// TwinCAT 3 PLC project Plc
// ProgramVersion: 3.1.4024.0
// libraries:
//   Tc2_Standard, * (Beckhoff Automation GmbH)
//   Tc2_System, * (Beckhoff Automation GmbH)
//   Tc3_Module, * (Beckhoff Automation GmbH)
// project tree:
//   / PlcTask.TcTTO
//   POUs/ MAIN.TcPOU, PRG_Testing.TcPOU
//   Utility/Actuator/ FB_Cylinder.TcPOU, FB_Cylinder_DoubleActing.TcPOU, FB_Cylinder_SingleActing.TcPOU
//   Utility/Sensor/ FB_Sensor_NC.TcPOU, FB_Sensor_NO.TcPOU
// real-time tasks:
//   TASK PlcTask: cycle T#10ms, priority 20, ADS port 350

CONFIGURATION Plc
    RESOURCE PLC ON TwinCAT3
        TASK PlcTask(INTERVAL := T#10ms, PRIORITY := 20);
        PROGRAM MAIN WITH PlcTask : MAIN;
    END_RESOURCE
END_CONFIGURATION

// ---- POUs/MAIN.TcPOU
PROGRAM MAIN
VAR
END_VAR

PRG_Testing();

END_PROGRAM

// ---- POUs/PRG_Testing.TcPOU
PROGRAM PRG_Testing
VAR
	fbCylinder_DoubleActing: FB_Cylinder_DoubleActing;
	fbCylinder_SingleActing: FB_Cylinder_SingleActing;
END_VAR


	fbCylinder_SingleActing(
	Start:= , 
	Extend:= , 
	Retract:= , 
	SensorExtended:= , 
	SensorRetracted:= , 
	EmergencyStop:= , 
	ExtendTime:= , 
	RetractTime:= , 
	Error=> , 
	ErrorCode=> , 
	Extend_RetractValve=> );
	
	fbCylinder_DoubleActing(
	Start:= , 
	Extend:= , 
	Retract:= , 
	SensorExtended:= , 
	SensorRetracted:= , 
	EmergencyStop:= , 
	ExtendTime:= , 
	RetractTime:= , 
	Error=> , 
	ErrorCode=> , 
	ExtendValve=> , 
	RetractValve=> );

END_PROGRAM

// ---- Utility/Actuator/FB_Cylinder_DoubleActing.TcPOU
FUNCTION_BLOCK FB_Cylinder_DoubleActing EXTENDS FB_Cylinder
VAR_INPUT
END_VAR
VAR_OUTPUT
    ExtendValve: BOOL;      // Valve output to extend the cylinder
    RetractValve: BOOL;     // Valve output to retract the cylinder	
END_VAR
VAR
END_VAR


	ExtendValve		:=	_ExtendValve;
	RetractValve	:=	_RetractValve;

END_FUNCTION_BLOCK

// ---- Utility/Actuator/FB_Cylinder.TcPOU
FUNCTION_BLOCK FB_Cylinder
VAR_INPUT
    Start: BOOL;                // Start signal
    Extend: BOOL;               // Extend signal
    Retract: BOOL;              // Retract signal
    SensorExtended: BOOL;       // Feedback from fully extended position sensor
    SensorRetracted: BOOL;      // Feedback from fully retracted position sensor
    EmergencyStop: BOOL;        // Emergency stop signal
    ExtendTime: TIME := T#5S;   // Time allowed to fully extend
    RetractTime: TIME := T#5S;  // Time allowed to fully retract
END_VAR

VAR_OUTPUT
    Error: BOOL;            // Error flag
    ErrorCode: INT;         // Error code for different fault conditions
END_VAR

VAR
    State: INT := 0;        // State variable for the state machine
    Timer: TON;             // Timer instance for timeouts
    _ExtendValve: BOOL;      // Valve output to extend the cylinder
    _RetractValve: BOOL;     // Valve output to retract the cylinder
END_VAR

	
	
	// State Machine Logic
	CASE State OF
		0: // Idle
			_ExtendValve := FALSE;
			_RetractValve := FALSE;
			Error := FALSE;
			ErrorCode := 0;
			
			IF EmergencyStop THEN
				State := 7; // Go to emergency stop state
			ELSIF Start THEN
				IF (Extend AND Retract) THEN
					Error := TRUE;
					ErrorCode := 1; // Invalid input (simultaneous Extend and Retract)
					State := 5; // Go to error state
				ELSIF Extend THEN
					IF NOT SensorExtended THEN
						State := 1; // Go to extend state if not already extended
					ELSE
						Error := TRUE;
						ErrorCode := 2; // Attempt to extend when already extended
						State := 5; // Go to error state
					END_IF
				ELSIF Retract THEN
					IF NOT SensorRetracted THEN
						State := 3; // Go to retract state if not already retracted
					ELSE
						Error := TRUE;
						ErrorCode := 3; // Attempt to retract when already retracted
						State := 5; // Go to error state
					END_IF
				END_IF
			END_IF
		
		1: // Extending
			_ExtendValve := TRUE;
			_RetractValve := FALSE;
			
			IF EmergencyStop THEN
				State := 7; // Go to emergency stop state
			ELSIF SensorExtended THEN
				State := 2; // Cylinder fully extended
			ELSE
				Timer(IN := TRUE, PT := ExtendTime); // Start timer for extension
				IF Timer.Q THEN
					Error := TRUE; // Timeout error
					ErrorCode := 4; // Failed to extend in time
					State := 5; // Go to error state
				END_IF
			END_IF
		
		2: // Extended
			_ExtendValve := FALSE;
			_RetractValve := FALSE;
			
			IF EmergencyStop THEN
				State := 7; // Go to emergency stop state
			ELSIF NOT Start THEN
				State := 0; // Return to Idle state when Start signal is released
			ELSIF Retract THEN
				IF NOT SensorRetracted THEN
					State := 3; // Go to retract state if not already retracted
				ELSE
					Error := TRUE;
					ErrorCode := 3; // Attempt to retract when already retracted
					State := 5; // Go to error state
				END_IF
			ELSIF (NOT SensorExtended AND NOT SensorRetracted) THEN
				State := 6; // Transition to stuck state if both sensors are off
			END_IF
		
		3: // Retracting
			_ExtendValve := FALSE;
			_RetractValve := TRUE;
			
			IF EmergencyStop THEN
				State := 7; // Go to emergency stop state
			ELSIF SensorRetracted THEN
				State := 4; // Cylinder fully retracted
			ELSE
				Timer(IN := TRUE, PT := RetractTime); // Start timer for retraction
				IF Timer.Q THEN
					Error := TRUE; // Timeout error
					ErrorCode := 5; // Failed to retract in time
					State := 5; // Go to error state
				END_IF
			END_IF
		
		4: // Retracted
			_ExtendValve := FALSE;
			_RetractValve := FALSE;
			
			IF EmergencyStop THEN
				State := 7; // Go to emergency stop state
			ELSIF NOT Start THEN
				State := 0; // Return to Idle state when Start signal is released
			ELSIF Extend THEN
				IF NOT SensorExtended THEN
					State := 1; // Go to extend state if not already extended
				ELSE
					Error := TRUE;
					ErrorCode := 2; // Attempt to extend when already extended
					State := 5; // Go to error state
				END_IF
			ELSIF (NOT SensorExtended AND NOT SensorRetracted) THEN
				State := 6; // Transition to stuck state if both sensors are off
			END_IF
		
		5: // Error
			_ExtendValve := FALSE;
			_RetractValve := FALSE;
			Error := TRUE;
			
			IF EmergencyStop THEN
				State := 7; // Go to emergency stop state
			ELSIF NOT Start THEN
				State := 0; // Return to Idle state
				Error := FALSE; // Reset error flag
				ErrorCode := 0; // Clear error code
			END_IF
		
		6: // Stuck in-between state
			_ExtendValve := FALSE;
			_RetractValve := FALSE;
			Error := TRUE;
			
			Timer(IN := TRUE, PT := T#10S); // 10-second stuck detection
			IF Timer.Q THEN
				ErrorCode := 6; // Cylinder stuck between positions
				State := 5; // Go to error state
			END_IF
			
			IF EmergencyStop THEN
				State := 7; // Go to emergency stop state
			ELSIF Extend THEN
				IF NOT SensorExtended THEN
					State := 1; // Go to extend state
				END_IF
			ELSIF Retract THEN
				IF NOT SensorRetracted THEN
					State := 3; // Go to retract state
				END_IF
			END_IF
		
		7: // Emergency stop state
			_ExtendValve := FALSE;     // Stop any motion immediately
			_RetractValve := FALSE;
			Error := TRUE;            // Signal an error
			ErrorCode := 7;           // Emergency stop error code
			
			// Stay in emergency state until EmergencyStop is cleared
			IF NOT EmergencyStop THEN
				State := 0; // Return to Idle state after emergency is cleared
				Error := FALSE;       // Clear error
				ErrorCode := 0;       // Clear error code
			END_IF
	END_CASE

END_FUNCTION_BLOCK

// ---- Utility/Actuator/FB_Cylinder_SingleActing.TcPOU
FUNCTION_BLOCK FB_Cylinder_SingleActing EXTENDS FB_Cylinder
VAR_INPUT
END_VAR
VAR_OUTPUT
	Extend_RetractValve: BOOL;	// 1: Valve output to extend the cylinder | 0: Valve output to retract the cylinder
END_VAR
VAR
END_VAR


	IF _ExtendValve AND (NOT _RetractValve) THEN
		Extend_RetractValve	:=	TRUE;
	ELSIF (NOT _ExtendValve) AND _RetractValve THEN
		Extend_RetractValve	:=	FALSE;
	ELSE
		Extend_RetractValve	:=	FALSE;
	END_IF

END_FUNCTION_BLOCK

// ---- Utility/Sensor/FB_Sensor_NC.TcPOU
FUNCTION_BLOCK FB_Sensor_NC
VAR_INPUT
END_VAR
VAR_OUTPUT
END_VAR
VAR
END_VAR

END_FUNCTION_BLOCK

// ---- Utility/Sensor/FB_Sensor_NO.TcPOU
FUNCTION_BLOCK FB_Sensor_NO
VAR_INPUT
END_VAR
VAR_OUTPUT
END_VAR
VAR
END_VAR

END_FUNCTION_BLOCK
